TYPE ST_LaudaReadCommands_ControlParameters :
STRUCT
END_STRUCT
END_TYPE

(* stored: Version 1.1.0.1, ProductVersion 3.1.4024.13
   DUT ST_LaudaReadCommands_ControlParameters: Id {705980ed-bc68-476c-b528-a865a7d42cd8} *)
